Staubli VAL3: PROG.dtx

num nChar = 89
num nFile = 2
progItem pEdit
  [0]
    InstrItem iEvent[2]
      [0]
        string sType = "PALLET"
        string sData = "prise"
      [1]
        string sType = "OUT"
        string sData = "bOut0>OFF AND bOut1>ON"
    string sID = "pick_place"
public string sItems
string sLine[100]
string sPathTemplate = "Disk://kernel/template/"
string sSession
string sTrajType
public string sWrite
